PROGRAM MAIN
VAR
	bTestBoolean :BOOL;
	nTestInt :INT;
	bTestBoolean2 :BOOL;
END_VAR

bTestBoolean :=TRUE;

bTestBoolean2 := bTestBoolean;

END_PROGRAM

(* stored: Version 1.1.0.1
   POU MAIN: Id {5f3a23e7-0d16-4948-b702-d7bd96dc9df1}, SpecialFunc None *)
